// TIA Portal V17 export
// export: Created 2025-05-22T06:01:04.4303613Z, ExportSetting WithDefaults, DisplayName Totally Integrated Automation Portal, DisplayVersion V17 Update 8, DisplayName TIA Portal Openness, DisplayVersion V17 Update 8, DisplayName TIA Portal Version Control Interface, DisplayVersion V17, DisplayName SINAMICS Startdrive Advanced, DisplayVersion V17 SP2, DisplayName SINAMICS Startdrive G110M, G120, G120C, G120D, G120P, G115D, DisplayVersion V17 SP2, DisplayName SINAMICS Startdrive G130, G150, S120, S150, SINAMICS MV, S210, DisplayVersion V17 SP2, DisplayName STEP 7 Professional, DisplayVersion V17 Update 8, DisplayName SINUMERIK ONE STEP 7 Toolbox, DisplayVersion V17 Update 12, DisplayName SINUMERIK ONE PLC Basic Program Plus, DisplayVersion V17 Update 12, DisplayName SINUMERIK 840D sl STEP 7 Toolbox, DisplayVersion V17 Update 12, DisplayName STEP 7 Safety, DisplayVersion V17 Update 6, DisplayName WinCC Advanced, DisplayVersion V17 Update 8
DATA_BLOCK "DB2109_UNIT_2_STATION_3_LIGHT"   // DB2109
{ DB_Accessible_From_OPC_UA := 'FALSE' }
VERSION : 0.1
// stored: AutoNumber false, DBAccessibleFromOPCUA false, DBAccessibleFromWebserver true, InstanceOfName FB2107_LIGHTS, InstanceOfType FB
"FB2107_LIGHTS"
   // VAR_INPUT
   //    GENERAL_MACHINE_LIGHT_OPTION : Bool;
   //    CIRCUIT_BRAKER_IN : Bool;
   //    LIGHT_ON_SELECTOR : Bool;
   //    MANUAL_REQ_LINE : Bool;
   //    SWITCH_ON_AUTO_REQ : Bool;
   //    SWITCH_OFF_AUTO_REQ : Bool;
   // END_VAR
   // VAR_OUTPUT
   //    LIGHTS_ON : Bool;
   //    HMI_LINE_ON_EXEC : Bool;
   //    HMI_LINE_OFF_EXEC : Bool;
   //    HMI_LINE_ON_STATUS : Bool;
   //    HMI_LINE_OFF_STATUS : Bool;
   // END_VAR
   // VAR
   //    SWITCH_ON_GENERAL_CONDITIONS : Bool;
   //    SWITCH_ON_INITIAL_CONDITIONS : Bool;
   //    SWITCH_ON_MANUAL_REQ : Bool;
   //    SWITCH_ON_GLOBAL_REQ : Bool;
   //    SWITCH_ON_COMMAND : Bool;
   //    SWITCH_ON : Bool;
   //    IN_SERVICE : Bool;
   //    SWITCH_OFF_GENERAL_CONDITIONS : Bool;
   //    SWITCH_OFF_INITIAL_CONDITIONS : Bool;
   //    SWITCH_OFF_MANUAL_REQ : Bool;
   //    SWITCH_OFF_GLOBAL_REQ : Bool;
   //    SWITCH_OFF_COMMAND : Bool;
   //    SWITCH_OFF : Bool;
   //    OUT_OF_SERVICE : Bool;
   //    SWITCH_ON_GLOBAL_REQUEST_AUX0 : Bool;
   //    SWITCH_ON_GLOBAL_REQUEST_AUX1 : Bool;
   //    SWITCH_ON_GLOBAL_REQUEST_AUX2 : Bool;
   //    SWITCH_ON_GLOBAL_REQUEST_AUX3 : Bool;
   //    SWITCH_OFF_GLOBAL_REQUEST_AUX1 : Bool;
   //    SWITCH_OFF_GLOBAL_REQUEST_AUX2 : Bool;
   //    SWITCH_OFF_DOORS_CLOSED_TIMER : IEC_TIMER;
   //    SWITCH_OFF_IN_SERVICE_DELAY_TIMER : IEC_TIMER;
   // END_VAR
BEGIN
END_DATA_BLOCK
